// TwinCAT 3 PLC project Untitled1
// ProgramVersion: 3.1.4023.0
// libraries:
//   Tc2_Standard, * (Beckhoff Automation GmbH)
//   Tc2_System, * (Beckhoff Automation GmbH)
//   Tc3_Module, * (Beckhoff Automation GmbH)
// project tree:
//   GVLs/ GVL.TcGVL
//   / PlcTask.TcTTO
//   POUs/ MAIN.TcPOU
// real-time tasks:
//   TASK PlcTask: cycle T#10ms, priority 20, ADS port 350
// I/O:
//   DEVICE Device 1 (Beckhoff CCAT)

CONFIGURATION Untitled1
    RESOURCE PLC ON TwinCAT3
        TASK PlcTask(INTERVAL := T#10ms, PRIORITY := 20);
        PROGRAM MAIN WITH PlcTask : MAIN;
    END_RESOURCE
END_CONFIGURATION

// ---- GVLs/GVL.TcGVL
{attribute 'qualified_only'}
VAR_GLOBAL
	QTY: DINT;
	T1_PT: TIME := T#1S;
	Word1: WORD;
	Word3: WORD;
	CSVWORD: ARRAY[0..1] OF WORD;
	Word2: WORD;
END_VAR

// ---- POUs/MAIN.TcPOU
PROGRAM MAIN
VAR
	T1: TON;
	T1_Q: BOOL;
END_VAR

T1_Q := NOT  T1.Q;
T1(IN:=T1_Q,PT:=GVL.T1_PT,Q=>);
IF T1.Q THEN
	GVL.QTY := GVL.QTY +100;
END_IF

END_PROGRAM
